PROGRAM MAIN
VAR
	fb_humiditysensor : FB_HumiditySensor;
	rHumidity : REAL;
	fb_cO2sensor : FB_CO2Sensor;
	rCO2Value : REAL;
	fb_temperaturesensor : FB_TemperatureSensor;
	rTemperature : REAL;
	fb_pressuresensor : FB_PressureSensor;
	rPressure : REAL;
END_VAR

fb_humiditysensor();
rHumidity := fb_humiditysensor.getHumidity;

fb_co2sensor();
rCO2Value := fb_co2sensor.getCO2Value;

fb_temperaturesensor();
rTemperature := fb_temperaturesensor.getTemperature;

fb_pressuresensor();
rPressure := fb_pressuresensor.getPressure;

END_PROGRAM

(* stored: Version 1.1.0.1, ProductVersion 3.1.4024.12
   POU MAIN: Id {53583b87-03a2-4d6c-8e12-0ff25b6d14c6}, SpecialFunc None *)
